FUNCTION_BLOCK Test_TStreamAdd_Read_T_MaxString EXTENDS TUnitTestBase
VAR
    Stream : TStream(StreamLength := 2);
    TestString : T_MaxString := '111111111 222222222 333333333 444444444 555555555 666666666 777777777 888888888 999999999 ';
END_VAR



Stream.Init(2);

Stream.Add_String(TestString);
    
Assertion.AssertEquals_UDINT(
    Expected := 91,
    Actual := Stream.Position,
    VariableName := 'Stream.Position');
    
Stream.Seek(0);

Assertion.AssertEquals_STRING(
    Expected := TestString,
    Actual := Stream.Read_String(),
    VariableName := 'Stream.Read_T_MaxString()');
    
Assertion.AssertEquals_UDINT(
    Expected := 91,
    Actual := Stream.Position,
    VariableName := 'Stream.Position');
    
    
TestFinished();

END_FUNCTION_BLOCK

(* stored: Version 1.1.0.1, ProductVersion 3.1.4024.4
   POU Test_TStreamAdd_Read_T_MaxString: Id {bbab0e0d-b28a-4d3d-a0a6-96ec30bda530}, SpecialFunc None *)
